FUNCTION F_softplus : lreal
VAR_INPUT
	x : LREAL;
END_VAR

F_softplus := log(exp(x)+1);

END_FUNCTION

(* stored: Version 1.1.0.1, ProductVersion 3.1.4024.12
   POU F_softplus: Id {595aca46-1dce-4de1-8177-d23da8043630}, SpecialFunc None *)
